TYPE ST_OPCUA_Server :
STRUCT
	sServerURL				: STRING;
	SessionConnectInfo		: ST_UASessionConnectInfo := (	tConnectTimeout			:= T#5S,
															tSessionTimeout 		:= T#1M,
															sApplicationName		:= '',
															eSecurityMode 			:= eUASecurityMsgMode_None,
															eSecurityPolicyUri	 	:= eUASecurityPolicy_None,
															eTransportProfileUri 	:= eUATransportProfileUri_UATcp);
	tTimeout            	: TIME := T#5M;
	nConnectionHdl			: DWORD;
END_STRUCT
END_TYPE

(* stored: Version 1.1.0.1, ProductVersion 3.1.4024.9
   DUT ST_OPCUA_Server: Id {219c0215-c4f5-466f-905d-335f835a3852} *)
